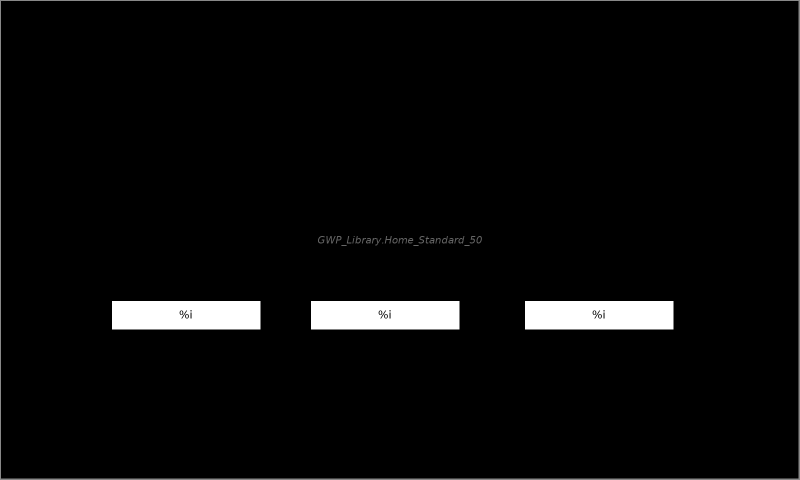
VISUALIZATION Home  // 800x480
    Frame (0,0 800x480)
        shows GWP_Library.Home_Standard_50(FB_Init_1 := Main.Init_0, FB_HS_Bool := Main.Anlageschalter)
    Rectangle (111,300 150x30), "%i"
    Rectangle (310,300 150x30), "%i"
    Rectangle (524,300 150x30), "%i"
END_VISUALIZATION

(* stored: Version 1.1.0.1, ProductVersion 3.1.4022.6
   Visu Home: Id {cf0d99aa-e151-45c6-a7fd-e762a0d2f343} *)
